TYPE TFError_WAM :
STRUCT
	Code 		: UINT; (*Codice di errore*)
	ExtraCode 	: UINT; (*Codice di errore EXTRA*)
END_STRUCT
END_TYPE

(* stored: Version 1.1.0.1, ProductVersion 3.1.4024.11
   DUT TFError_WAM: Id {24f63ef1-ddd5-449a-abbf-bbaf750a2235} *)
